SUBAPPLICATION PositionSensor (* Subapplication Type *)
  (* Standard: 61499-2 *)
  (* Version 1.0, 2025-03-21, AK123700 *)
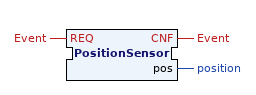
  EVENT_INPUT
    REQ; (* Normal Execution Request *)
  END_EVENT
  EVENT_OUTPUT
    CNF; (* Execution Confirmation *)
  END_EVENT
  VAR_OUTPUT
    pos : position;
  END_VAR
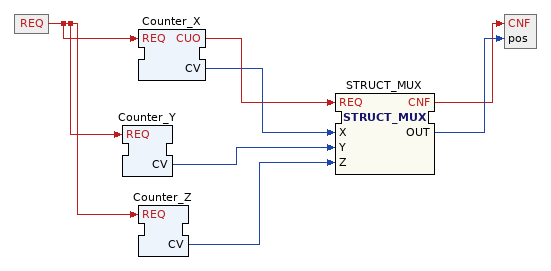
  FBS
    STRUCT_MUX : STRUCT_MUX; {SET_ATTRIBUTE(StructuredType, position)}
  END_FBS
  SUBAPPLICATION Counter_X
    EVENT_INPUT
      REQ;
    END_EVENT
    EVENT_OUTPUT
      CUO;
    END_EVENT
    VAR_OUTPUT
      CV : UINT;
    END_VAR
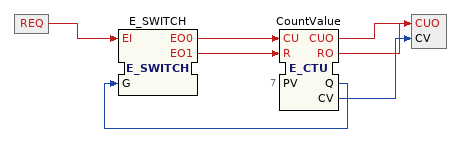
    FBS
      E_SWITCH : E_SWITCH;
      CountValue : E_CTU(PV := 7);
    END_FBS
    EVENT_CONNECTIONS
      E_SWITCH.EO0 TO CountValue.CU;
      E_SWITCH.EO1 TO CountValue.R;
      REQ TO E_SWITCH.EI;
      CountValue.CUO TO CUO;
      CountValue.RO TO CUO;
    END_CONNECTIONS
    DATA_CONNECTIONS
      CountValue.Q TO E_SWITCH.G;
      CountValue.CV TO CV;
    END_CONNECTIONS
  END_SUBAPPLICATION
  SUBAPPLICATION Counter_Y
    EVENT_INPUT
      REQ;
    END_EVENT
    VAR_OUTPUT
      CV : UINT;
    END_VAR
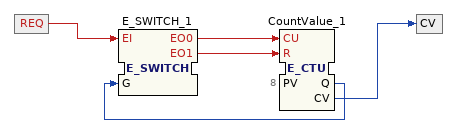
    FBS
      CountValue_1 : E_CTU(PV := 8);
      E_SWITCH_1 : E_SWITCH;
    END_FBS
    EVENT_CONNECTIONS
      E_SWITCH_1.EO0 TO CountValue_1.CU;
      E_SWITCH_1.EO1 TO CountValue_1.R;
      REQ TO E_SWITCH_1.EI;
    END_CONNECTIONS
    DATA_CONNECTIONS
      CountValue_1.Q TO E_SWITCH_1.G;
      CountValue_1.CV TO CV;
    END_CONNECTIONS
  END_SUBAPPLICATION
  SUBAPPLICATION Counter_Z
    EVENT_INPUT
      REQ;
    END_EVENT
    VAR_OUTPUT
      CV : UINT;
    END_VAR
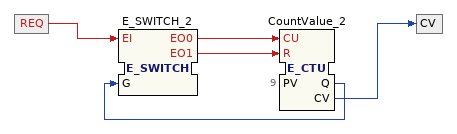
    FBS
      CountValue_2 : E_CTU(PV := 9);
      E_SWITCH_2 : E_SWITCH;
    END_FBS
    EVENT_CONNECTIONS
      E_SWITCH_2.EO0 TO CountValue_2.CU;
      E_SWITCH_2.EO1 TO CountValue_2.R;
      REQ TO E_SWITCH_2.EI;
    END_CONNECTIONS
    DATA_CONNECTIONS
      CountValue_2.Q TO E_SWITCH_2.G;
      CountValue_2.CV TO CV;
    END_CONNECTIONS
  END_SUBAPPLICATION
  EVENT_CONNECTIONS
    REQ TO Counter_X.REQ;
    REQ TO Counter_Y.REQ;
    REQ TO Counter_Z.REQ;
    Counter_X.CUO TO STRUCT_MUX.REQ;
    STRUCT_MUX.CNF TO CNF;
  END_CONNECTIONS
  DATA_CONNECTIONS
    STRUCT_MUX.OUT TO pos;
    Counter_X.CV TO STRUCT_MUX.X;
    Counter_Y.CV TO STRUCT_MUX.Y;
    Counter_Z.CV TO STRUCT_MUX.Z;
  END_CONNECTIONS
END_SUBAPPLICATION
